VAR_GLOBAL
	
Axis1 : AXIS_REF;
stAxis1	:	stAxisInterface;


END_VAR

(* stored: Version 1.1.0.1, ProductVersion 3.1.4024.4
   GVL GVL_Axis: Id {fc0173b8-b65d-42c4-afe5-a310bf3ca9e3} *)
